// TIA Portal V17 export
// export: Created 2022-05-07T16:38:46.7545648Z, ExportSetting WithDefaults, DisplayName Totally Integrated Automation Portal, DisplayVersion V17 Update 3, DisplayName TIA Portal Openness, DisplayVersion V17 Update 3, DisplayName TIA Portal Version Control Interface, DisplayVersion V17, DisplayName TIA Portal Test Suite Advanced, DisplayVersion V17 Update 1, DisplayName SINAMICS Startdrive Advanced, DisplayVersion V17 Update2, DisplayName SINAMICS Startdrive G130, G150, S120, S150, SINAMICS MV, S210, DisplayVersion V17 Update2, DisplayName SINAMICS Startdrive G110M, G120, G120C, G120D, G120P, G115D, DisplayVersion V17 Update2, DisplayName STEP 7 Professional, DisplayVersion V17 Update 3, DisplayName STEP 7 Safety, DisplayVersion V17, DisplayName WinCC UA Professional, DisplayVersion V17 Update 3
DATA_BLOCK "FB_CICLO_DB"   // DB11
VERSION : 0.1
// stored: AutoNumber true, DBAccessibleFromOPCUA true, InstanceOfName FB_CICLO_GEN, InstanceOfType FB
"FB_CICLO_GEN"
   // VAR_OUTPUT
   //    fase : Int;
   // END_VAR
   // VAR
   //    condOkStartCiclo { S7_SetPoint := 'True'} : Bool;
   //    T10 { S7_SetPoint := 'True'} : TON_TIME;
   //    T20 { S7_SetPoint := 'True'} : TON_TIME;
   //    T30 { S7_SetPoint := 'True'} : TON_TIME;
   //    T40 { S7_SetPoint := 'True'} : TON_TIME;
   //    T50 { S7_SetPoint := 'True'} : TON_TIME;
   //    T60 { S7_SetPoint := 'True'} : TON_TIME;
   //    T70 { S7_SetPoint := 'True'} : TON_TIME;
   //    T75 { S7_SetPoint := 'True'} : TON_TIME;
   //    T80 { S7_SetPoint := 'True'} : TON_TIME;
   //    T90 { S7_SetPoint := 'True'} : TON_TIME;
   //    T100 { S7_SetPoint := 'True'} : TON_TIME;
   //    TcicloPrec { S7_SetPoint := 'True'} : Int;
   //    TCicloAtt : Int;
   //    appQuotaStartStrappi : Real;
   //    FNStartCiclo : Bool;
   //    AppFNStartCiclo : Bool;
   //    FPClok01s : Bool;
   //    AppFPClok01s : Bool;
   //    appComandoIndietroME : Bool;
   // END_VAR
BEGIN
END_DATA_BLOCK
